(* IEC 61131-3 sources: CodesysTest/alpha/export/FBs/Components/Load Plate/FB_BaseLoadPlate.pou/Shaking.prop, 1 file *)

(* ---- Get.pm.st ---- *)
(*#-#-#-#-#-#-#-#-#-#---Declaration---#-#-#-#-#-#-#-#-#-#-#-#-#*)

VAR
END_VAR
(*#-#-#-#-#-#-#-#-#-#---Implementation---#-#-#-#-#-#-#-#-#-#-#-#-#*)

Shaking := _shake OR _state <> LOAD_PLATE_STATE.Idle;
